// TIA Portal V17 export
// export: Created 2024-08-07T21:44:08.5756409Z, ExportSetting WithDefaults, DisplayName Totally Integrated Automation Portal, DisplayVersion V17 Update 7, DisplayName TIA Portal Openness, DisplayVersion V17 Update 7, DisplayName TIA Portal Version Control Interface, DisplayVersion V17, DisplayName SINAMICS Startdrive Advanced, DisplayVersion V17 SP2, DisplayName SINAMICS Startdrive G110M, G120, G120C, G120D, G120P, G115D, DisplayVersion V17 SP2, DisplayName SINAMICS Startdrive G130, G150, S120, S150, SINAMICS MV, S210, DisplayVersion V17 SP2, DisplayName STEP 7 Professional, DisplayVersion V17 Update 7, DisplayName STEP 7 Safety, DisplayVersion V17 Update 6, DisplayName WinCC Advanced / Unified PC, DisplayVersion V17 Update 7
DATA_BLOCK "safety_signals"   // DB2, F_DB
{ S7_Optimized_Access := 'TRUE' }
VERSION : 0.1
// stored: AutoNumber true, DBAccessibleFromOPCUA true, DBAccessibleFromWebserver true
   VAR
      estopok : Bool := FALSE;
      lightBarrierOk : Bool := FALSE;
      tableInPosition : Bool := FALSE;
      contactorsOk : Bool := FALSE;
      maintenanceDoorsClosed : Bool := FALSE;
      operateRobot1 : Bool := FALSE;
      serviceMode : Bool := FALSE;
      CoversClosed : Bool := FALSE;   // Emergency buttons and covers closed
      "3L+" : Bool := TRUE;   // emergency stop
      "4L+" : Bool := TRUE;   // emergency stop + service doors
      "5L+" : Bool := FALSE;   // emergency stop + service doors + light curtain
      serviceModeEnabled : Bool := FALSE;
      ACK_REI_Req : Bool := FALSE;
      RobotKeyNecessary : Bool := FALSE;
      Clock_1Hz : Bool := TRUE;
      doorUnlocked : Bool := FALSE;
   END_VAR
BEGIN
END_DATA_BLOCK
